// SIMATIC S7-200 project (STEP 7-Micro/WIN), CPU 224 REL 01.22

ORGANIZATION_BLOCK MAIN:OB1
TITLE=POU Comment
BEGIN
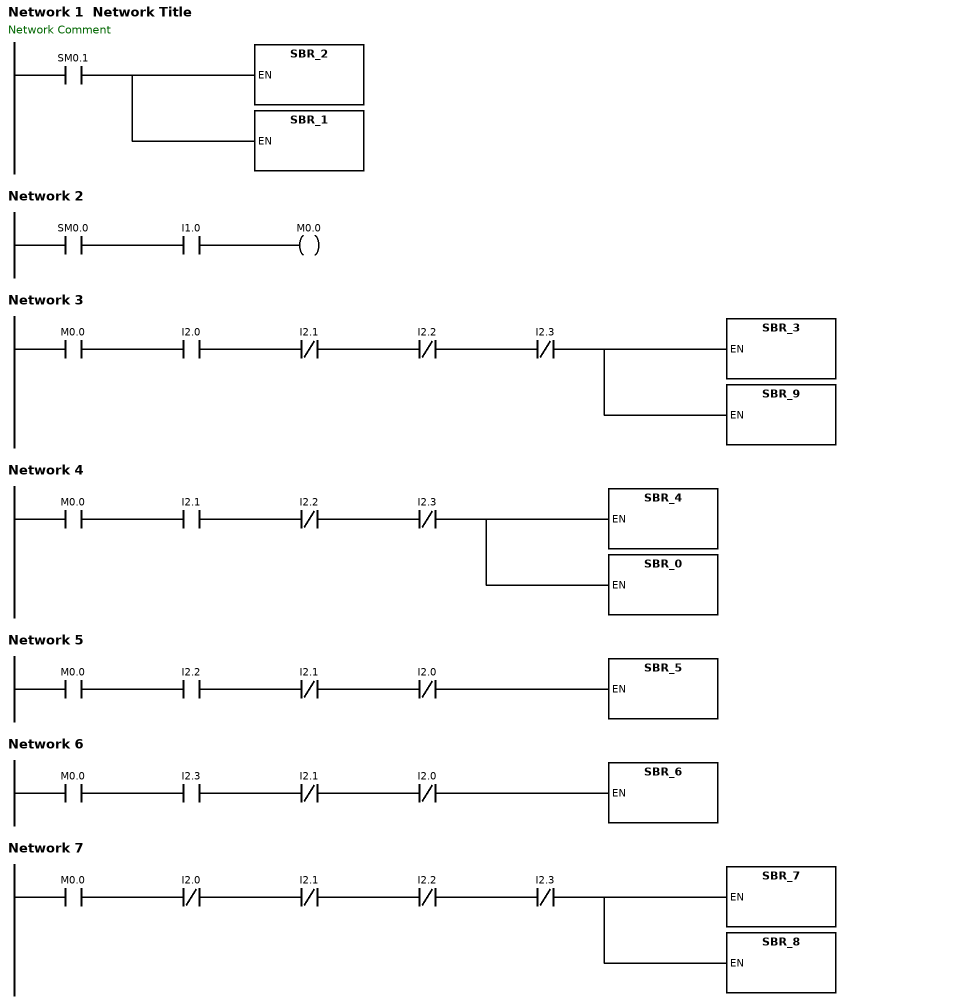
Network 1 // Network Title
// Network Comment
LD     SM0.1
CALL   SBR_2:SBR2
CALL   SBR_1:SBR1
Network 2
LD     SM0.0
A      I1.0
=      M0.0
Network 3
LD     M0.0
A      I2.0
AN     I2.1
AN     I2.2
AN     I2.3
CALL   SBR_3:SBR3
CALL   SBR_9:SBR9
Network 4
LD     M0.0
A      I2.1
AN     I2.2
AN     I2.3
CALL   SBR_4:SBR4
CALL   SBR_0:SBR0
Network 5
LD     M0.0
A      I2.2
AN     I2.1
AN     I2.0
CALL   SBR_5:SBR5
Network 6
LD     M0.0
A      I2.3
AN     I2.1
AN     I2.0
CALL   SBR_6:SBR6
Network 7
LD     M0.0
AN     I2.0
AN     I2.1
AN     I2.2
AN     I2.3
CALL   SBR_7:SBR7
CALL   SBR_8:SBR8
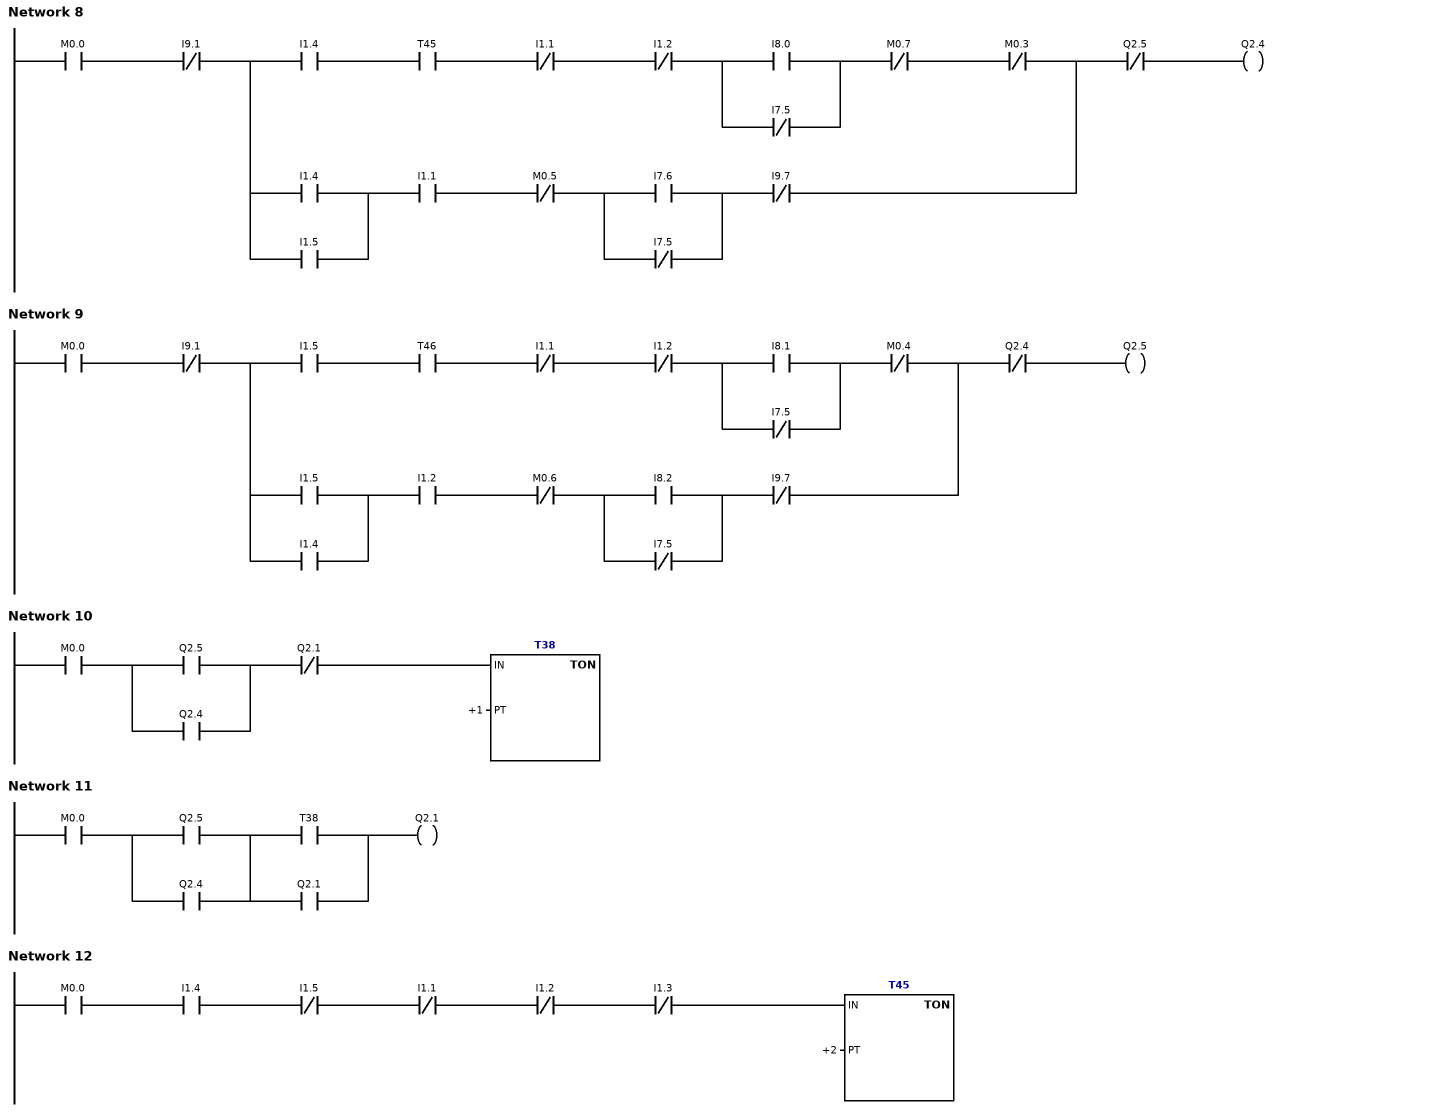
Network 8
LD     M0.0
AN     I9.1
LD     I1.4
A      T45
AN     I1.1
AN     I1.2
LD     I8.0
ON     I7.5
ALD
AN     M0.7
AN     M0.3
LD     I1.4
O      I1.5
A      I1.1
AN     M0.5
LD     I7.6
ON     I7.5
ALD
AN     I9.7
OLD
ALD
AN     Q2.5
=      Q2.4
Network 9
LD     M0.0
AN     I9.1
LD     I1.5
A      T46
AN     I1.1
AN     I1.2
LD     I8.1
ON     I7.5
ALD
AN     M0.4
LD     I1.5
O      I1.4
A      I1.2
AN     M0.6
LD     I8.2
ON     I7.5
ALD
AN     I9.7
OLD
ALD
AN     Q2.4
=      Q2.5
Network 10
LD     M0.0
LD     Q2.5
O      Q2.4
ALD
AN     Q2.1
TON    T38, +1
Network 11
LD     M0.0
LD     Q2.5
O      Q2.4
ALD
LD     T38
O      Q2.1
ALD
=      Q2.1
Network 12
LD     M0.0
A      I1.4
AN     I1.5
AN     I1.1
AN     I1.2
AN     I1.3
TON    T45, +2
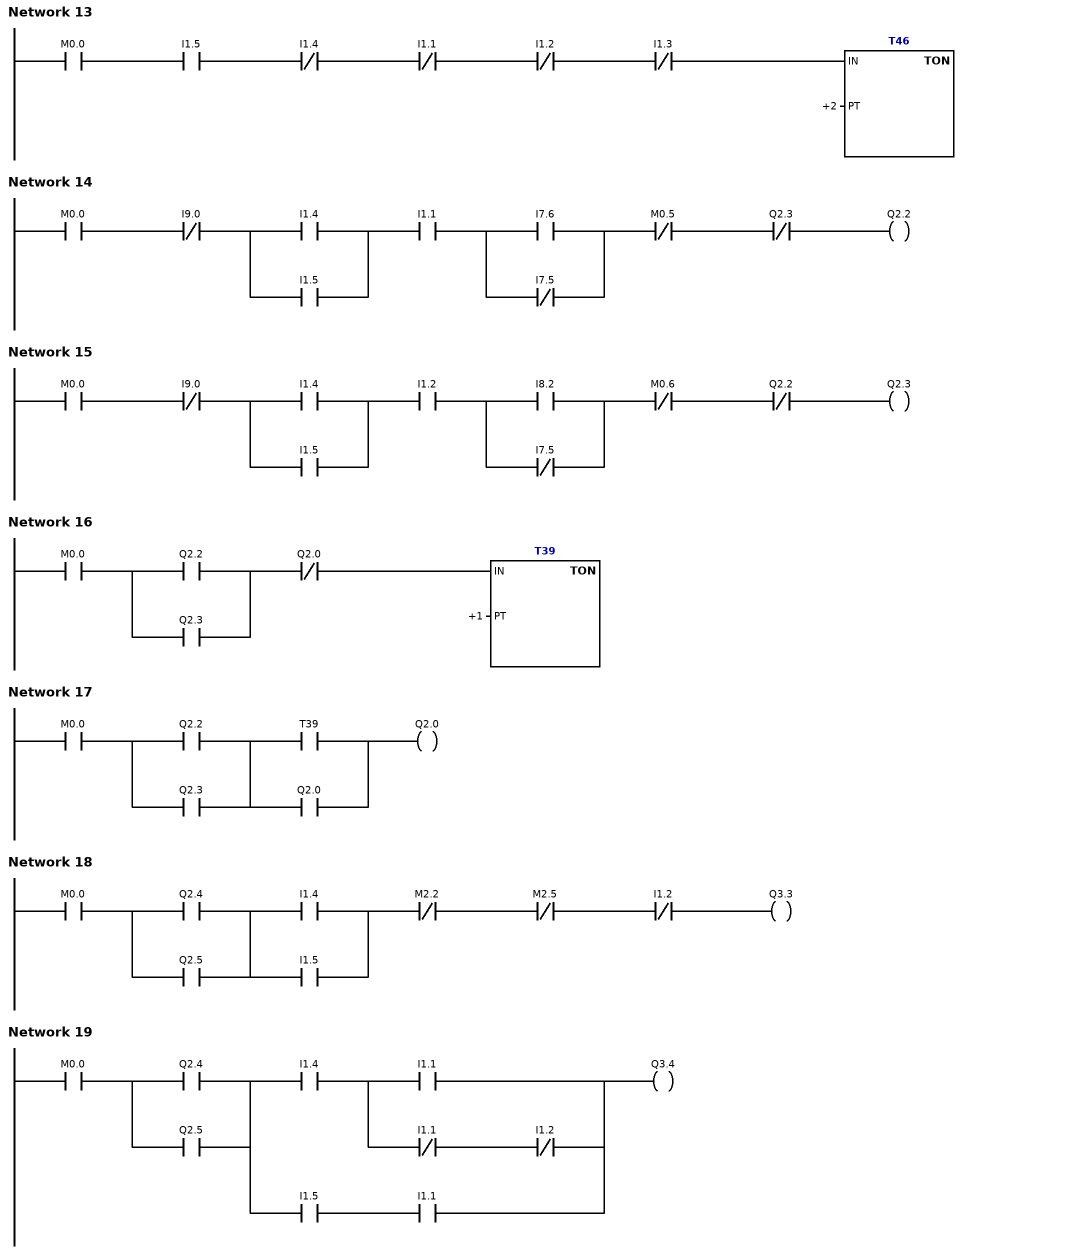
Network 13
LD     M0.0
A      I1.5
AN     I1.4
AN     I1.1
AN     I1.2
AN     I1.3
TON    T46, +2
Network 14
LD     M0.0
AN     I9.0
LD     I1.4
O      I1.5
ALD
A      I1.1
LD     I7.6
ON     I7.5
ALD
AN     M0.5
AN     Q2.3
=      Q2.2
Network 15
LD     M0.0
AN     I9.0
LD     I1.4
O      I1.5
ALD
A      I1.2
LD     I8.2
ON     I7.5
ALD
AN     M0.6
AN     Q2.2
=      Q2.3
Network 16
LD     M0.0
LD     Q2.2
O      Q2.3
ALD
AN     Q2.0
TON    T39, +1
Network 17
LD     M0.0
LD     Q2.2
O      Q2.3
ALD
LD     T39
O      Q2.0
ALD
=      Q2.0
Network 18
LD     M0.0
LD     Q2.4
O      Q2.5
ALD
LD     I1.4
O      I1.5
ALD
AN     M2.2
AN     M2.5
AN     I1.2
=      Q3.3
Network 19
LD     M0.0
LD     Q2.4
O      Q2.5
ALD
LD     I1.4
LD     I1.1
LDN    I1.1
AN     I1.2
OLD
ALD
LD     I1.5
A      I1.1
OLD
ALD
=      Q3.4
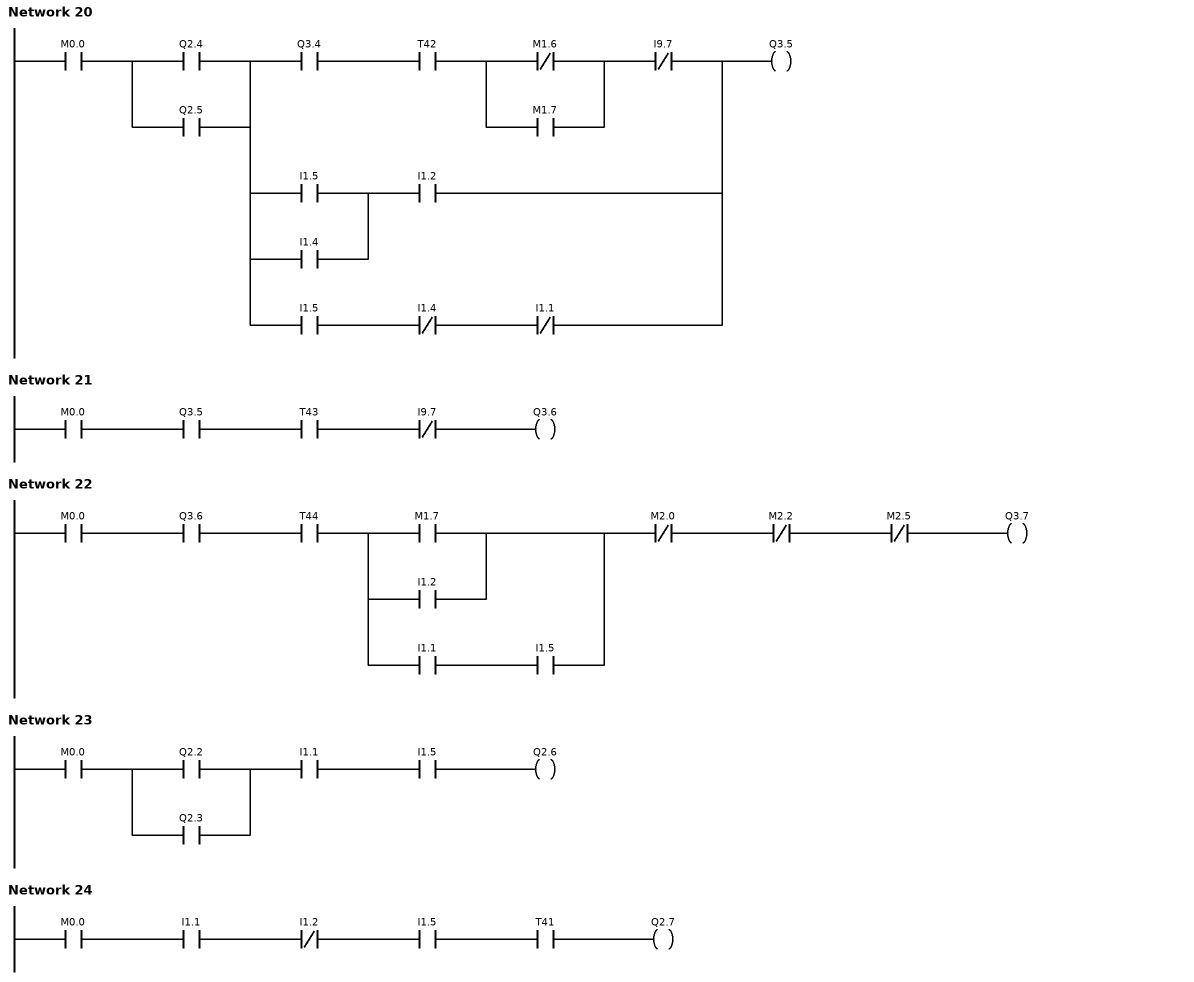
Network 20
LD     M0.0
LD     Q2.4
O      Q2.5
ALD
LD     Q3.4
A      T42
LDN    M1.6
O      M1.7
ALD
AN     I9.7
LD     I1.5
O      I1.4
A      I1.2
OLD
LD     I1.5
AN     I1.4
AN     I1.1
OLD
ALD
=      Q3.5
Network 21
LD     M0.0
A      Q3.5
A      T43
AN     I9.7
=      Q3.6
Network 22
LD     M0.0
A      Q3.6
A      T44
LD     M1.7
O      I1.2
LD     I1.1
A      I1.5
OLD
ALD
AN     M2.0
AN     M2.2
AN     M2.5
=      Q3.7
Network 23
LD     M0.0
LD     Q2.2
O      Q2.3
ALD
A      I1.1
A      I1.5
=      Q2.6
Network 24
LD     M0.0
A      I1.1
AN     I1.2
A      I1.5
A      T41
=      Q2.7
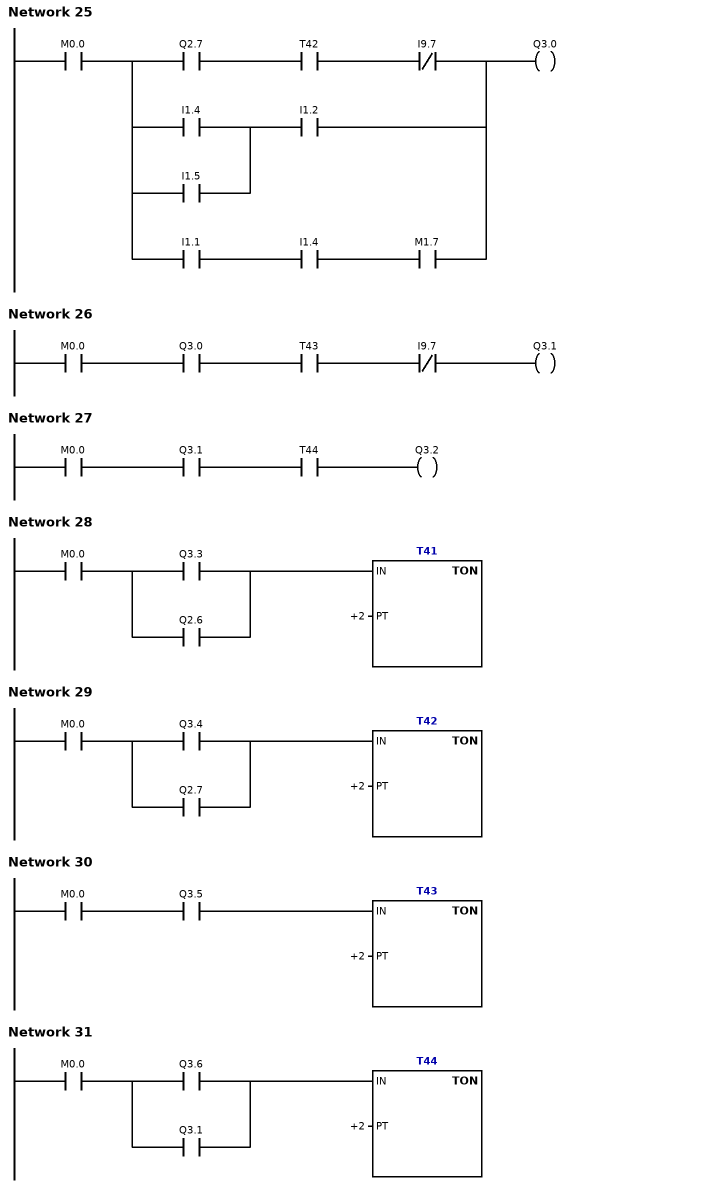
Network 25
LD     M0.0
LD     Q2.7
A      T42
AN     I9.7
LD     I1.4
O      I1.5
A      I1.2
OLD
LD     I1.1
A      I1.4
A      M1.7
OLD
ALD
=      Q3.0
Network 26
LD     M0.0
A      Q3.0
A      T43
AN     I9.7
=      Q3.1
Network 27
LD     M0.0
A      Q3.1
A      T44
=      Q3.2
Network 28
LD     M0.0
LD     Q3.3
O      Q2.6
ALD
TON    T41, +2
Network 29
LD     M0.0
LD     Q3.4
O      Q2.7
ALD
TON    T42, +2
Network 30
LD     M0.0
A      Q3.5
TON    T43, +2
Network 31
LD     M0.0
LD     Q3.6
O      Q3.1
ALD
TON    T44, +2
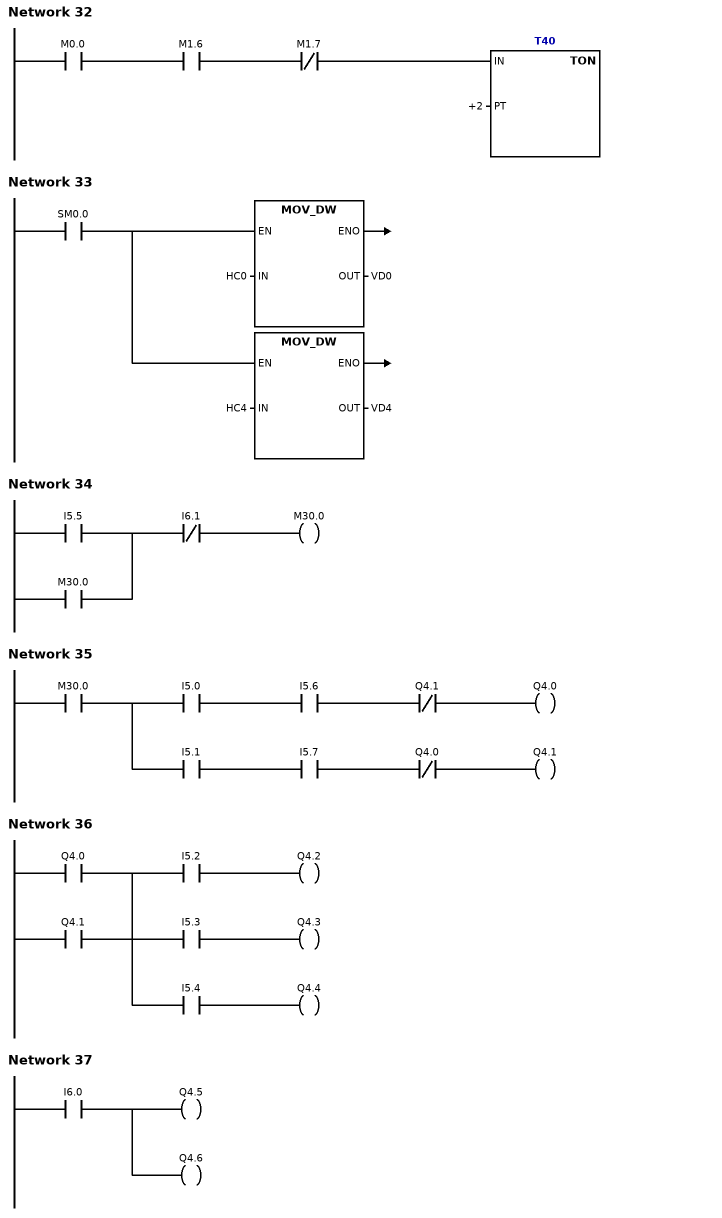
Network 32
LD     M0.0
A      M1.6
AN     M1.7
TON    T40, +2
Network 33
LD     SM0.0
MOVD   HC0, VD0
MOVD   HC4, VD4
Network 34
LD     I5.5
O      M30.0
AN     I6.1
=      M30.0
Network 35
LD     M30.0
LPS
A      I5.0
A      I5.6
AN     Q4.1
=      Q4.0
LPP
A      I5.1
A      I5.7
AN     Q4.0
=      Q4.1
Network 36
LD     Q4.0
O      Q4.1
LPS
A      I5.2
=      Q4.2
LRD
A      I5.3
=      Q4.3
LPP
A      I5.4
=      Q4.4
Network 37
LD     I6.0
=      Q4.5
=      Q4.6
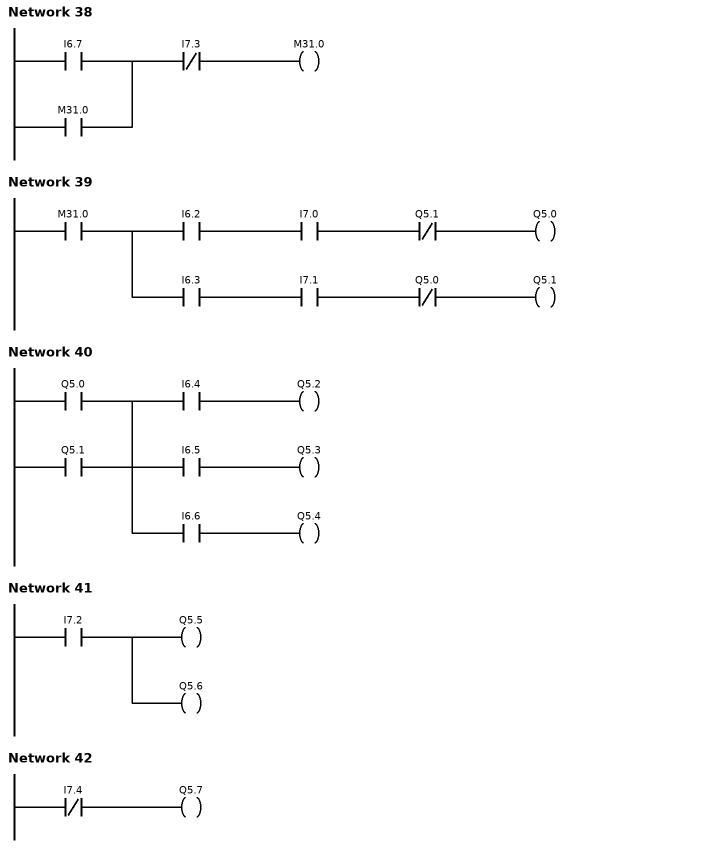
Network 38
LD     I6.7
O      M31.0
AN     I7.3
=      M31.0
Network 39
LD     M31.0
LPS
A      I6.2
A      I7.0
AN     Q5.1
=      Q5.0
LPP
A      I6.3
A      I7.1
AN     Q5.0
=      Q5.1
Network 40
LD     Q5.0
O      Q5.1
LPS
A      I6.4
=      Q5.2
LRD
A      I6.5
=      Q5.3
LPP
A      I6.6
=      Q5.4
Network 41
LD     I7.2
=      Q5.5
=      Q5.6
Network 42
LDN    I7.4
=      Q5.7
END_ORGANIZATION_BLOCK

SUBROUTINE_BLOCK SBR_0:SBR0
TITLE=POU Comment
BEGIN
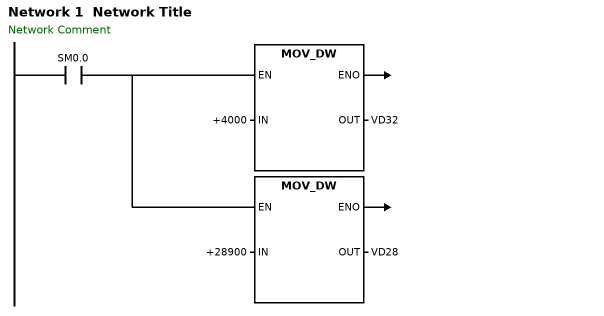
Network 1 // Network Title
// Network Comment
// (network saved uncompiled; LAD cells follow)
// row 0: c0 -| |- SM0.0 v  c1 --  c2 [MOV_DW EN:=power@row0, IN:=+4000, ENO=>power, OUT=>VD32]  c3 ->
// row 1: c0 ^v  c2 [box]
// row 2: c0 ^  c1 --  c2 [MOV_DW EN:=power@row2, IN:=+28900, ENO=>power, OUT=>VD28]  c3 ->
// row 3: c2 [box]
END_SUBROUTINE_BLOCK

SUBROUTINE_BLOCK SBR_1:SBR1
TITLE=
BEGIN
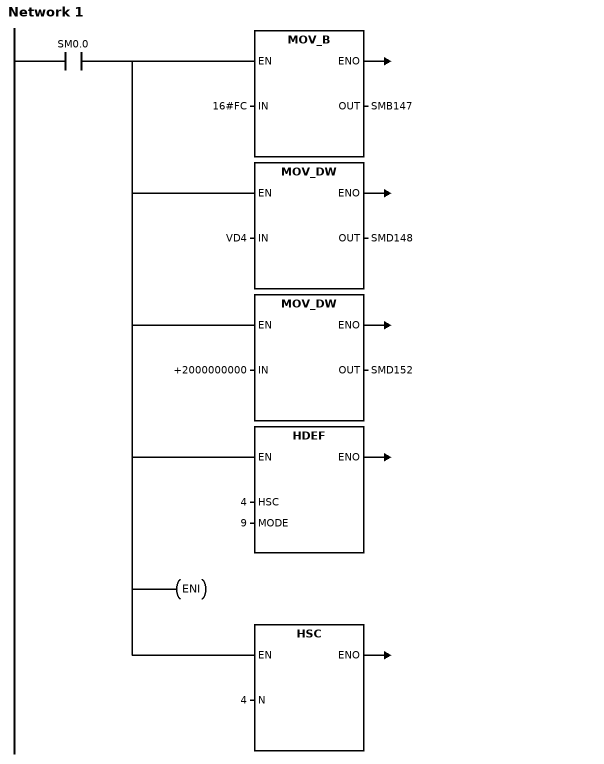
Network 1
// (network saved uncompiled; LAD cells follow)
// row 0: c0 -| |- SM0.0 v  c1 --  c2 [MOV_B EN:=power@row0, IN:=16#FC, ENO=>power, OUT=>SMB147]  c3 ->
// row 1: c0 ^v  c2 [box]
// row 2: c0 ^v  c1 --  c2 [MOV_DW EN:=power@row2, IN:=VD4, ENO=>power, OUT=>SMD148]  c3 ->
// row 3: c0 ^v  c2 [box]
// row 4: c0 ^v  c1 --  c2 [MOV_DW EN:=power@row4, IN:=+2000000000, ENO=>power, OUT=>SMD152]  c3 ->
// row 5: c0 ^v  c2 [box]
// row 6: c0 ^v  c1 --  c2 [HDEF EN:=power@row6, HSC:=4, MODE:=9, ENO=>power]  c3 ->
// row 7: c0 ^v  c2 [box]
// row 8: c0 ^v  c1 -(ENI)
// row 9: c0 ^  c1 --  c2 [HSC EN:=power@row9, N:=4, ENO=>power]  c3 ->
// row 10: c2 [box]
END_SUBROUTINE_BLOCK

SUBROUTINE_BLOCK SBR_2:SBR2
TITLE=
BEGIN
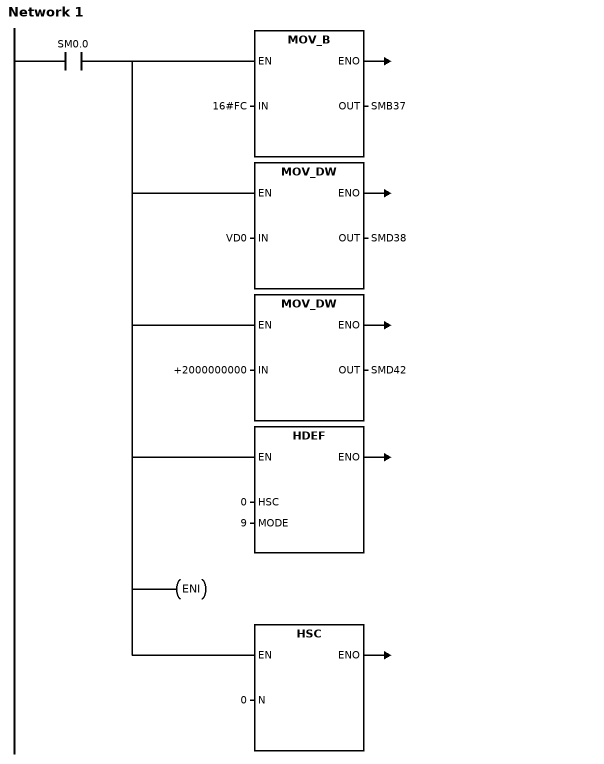
Network 1
// (network saved uncompiled; LAD cells follow)
// row 0: c0 -| |- SM0.0 v  c1 --  c2 [MOV_B EN:=power@row0, IN:=16#FC, ENO=>power, OUT=>SMB37]  c3 ->
// row 1: c0 ^v  c2 [box]
// row 2: c0 ^v  c1 --  c2 [MOV_DW EN:=power@row2, IN:=VD0, ENO=>power, OUT=>SMD38]  c3 ->
// row 3: c0 ^v  c2 [box]
// row 4: c0 ^v  c1 --  c2 [MOV_DW EN:=power@row4, IN:=+2000000000, ENO=>power, OUT=>SMD42]  c3 ->
// row 5: c0 ^v  c2 [box]
// row 6: c0 ^v  c1 --  c2 [HDEF EN:=power@row6, HSC:=0, MODE:=9, ENO=>power]  c3 ->
// row 7: c0 ^v  c2 [box]
// row 8: c0 ^v  c1 -(ENI)
// row 9: c0 ^  c1 --  c2 [HSC EN:=power@row9, N:=0, ENO=>power]  c3 ->
// row 10: c2 [box]
END_SUBROUTINE_BLOCK

SUBROUTINE_BLOCK SBR_3:SBR3
TITLE=
BEGIN
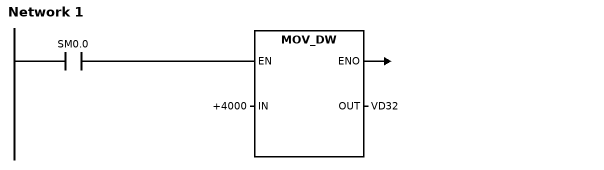
Network 1
// (network saved uncompiled; LAD cells follow)
// row 0: c0 -| |- SM0.0  c1 --  c2 [MOV_DW EN:=power@row0, IN:=+4000, ENO=>power, OUT=>VD32]  c3 ->
// row 1: c2 [box]
END_SUBROUTINE_BLOCK

SUBROUTINE_BLOCK SBR_4:SBR4
TITLE=
BEGIN
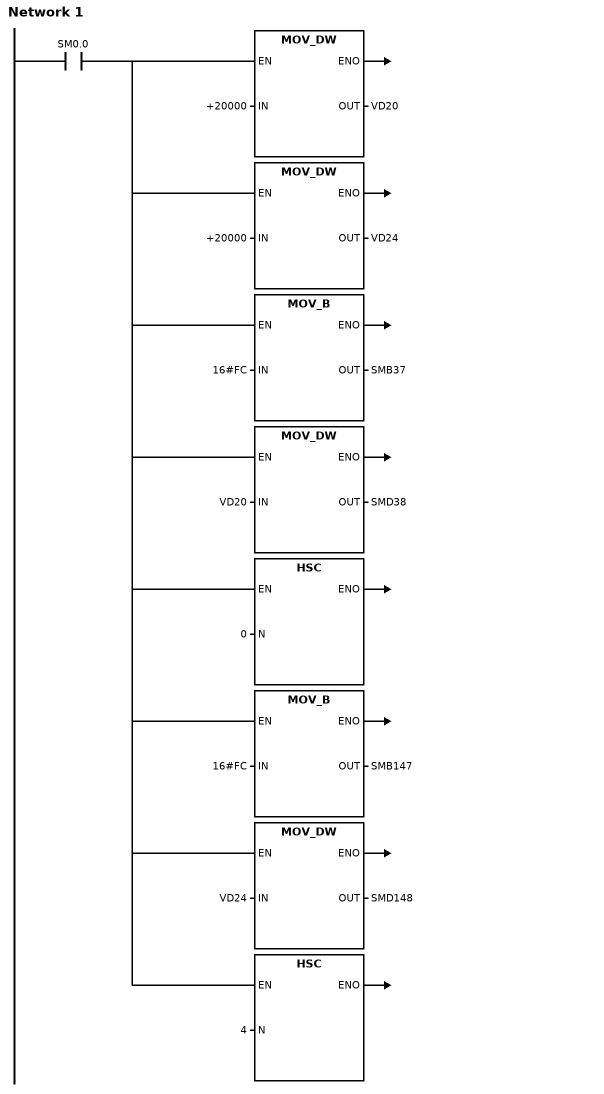
Network 1
// (network saved uncompiled; LAD cells follow)
// row 0: c0 -| |- SM0.0 v  c1 --  c2 [MOV_DW EN:=power@row0, IN:=+20000, ENO=>power, OUT=>VD20]  c3 ->
// row 1: c0 ^v  c2 [box]
// row 2: c0 ^v  c1 --  c2 [MOV_DW EN:=power@row2, IN:=+20000, ENO=>power, OUT=>VD24]  c3 ->
// row 3: c0 ^v  c2 [box]
// row 4: c0 ^v  c1 --  c2 [MOV_B EN:=power@row4, IN:=16#FC, ENO=>power, OUT=>SMB37]  c3 ->
// row 5: c0 ^v  c2 [box]
// row 6: c0 ^v  c1 --  c2 [MOV_DW EN:=power@row6, IN:=VD20, ENO=>power, OUT=>SMD38]  c3 ->
// row 7: c0 ^v  c2 [box]
// row 8: c0 ^v  c1 --  c2 [HSC EN:=power@row8, N:=0, ENO=>power]  c3 ->
// row 9: c0 ^v  c2 [box]
// row 10: c0 ^v  c1 --  c2 [MOV_B EN:=power@row10, IN:=16#FC, ENO=>power, OUT=>SMB147]  c3 ->
// row 11: c0 ^v  c2 [box]
// row 12: c0 ^v  c1 --  c2 [MOV_DW EN:=power@row12, IN:=VD24, ENO=>power, OUT=>SMD148]  c3 ->
// row 13: c0 ^v  c2 [box]
// row 14: c0 ^  c1 --  c2 [HSC EN:=power@row14, N:=4, ENO=>power]  c3 ->
// row 15: c2 [box]
END_SUBROUTINE_BLOCK

SUBROUTINE_BLOCK SBR_5:SBR5
TITLE=
BEGIN
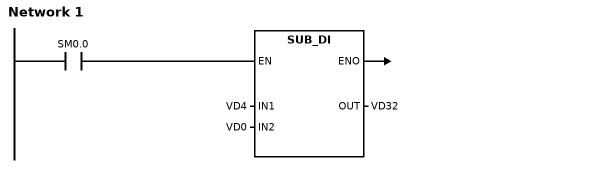
Network 1
// (network saved uncompiled; LAD cells follow)
// row 0: c0 -| |- SM0.0  c1 --  c2 [SUB_DI EN:=power@row0, IN1:=VD4, IN2:=VD0, ENO=>power, OUT=>VD32]  c3 ->
// row 1: c2 [box]
END_SUBROUTINE_BLOCK

SUBROUTINE_BLOCK SBR_6:SBR6
TITLE=
BEGIN
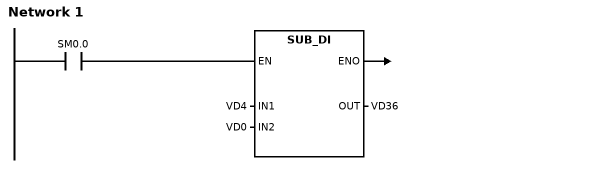
Network 1
// (network saved uncompiled; LAD cells follow)
// row 0: c0 -| |- SM0.0  c1 --  c2 [SUB_DI EN:=power@row0, IN1:=VD4, IN2:=VD0, ENO=>power, OUT=>VD36]  c3 ->
// row 1: c2 [box]
END_SUBROUTINE_BLOCK

SUBROUTINE_BLOCK SBR_7:SBR7
TITLE=
BEGIN
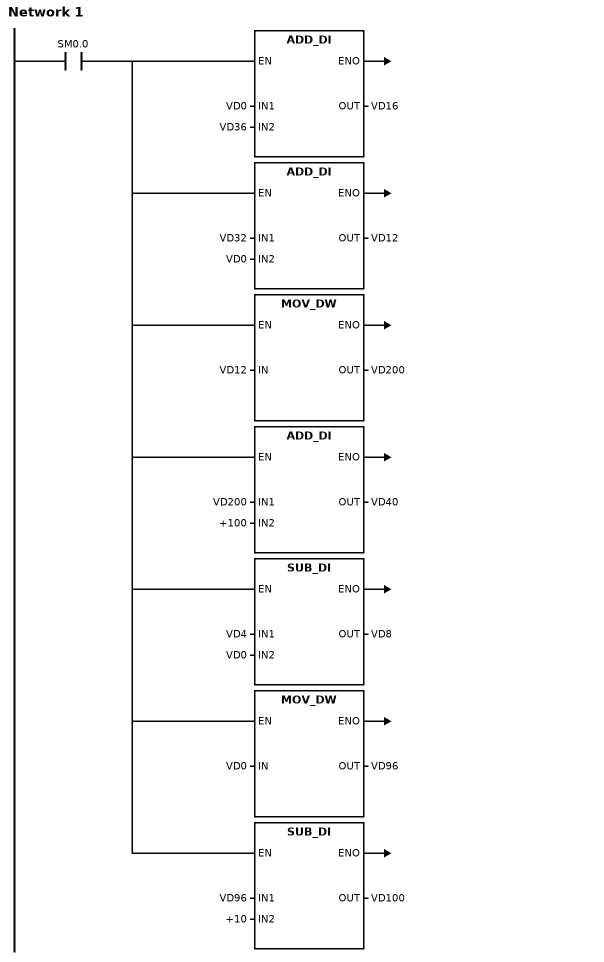
Network 1
// (network saved uncompiled; LAD cells follow)
// row 0: c0 -| |- SM0.0 v  c1 --  c2 [ADD_DI EN:=power@row0, IN1:=VD0, IN2:=VD36, ENO=>power, OUT=>VD16]  c3 ->
// row 1: c0 ^v  c2 [box]
// row 2: c0 ^v  c1 --  c2 [ADD_DI EN:=power@row2, IN1:=VD32, IN2:=VD0, ENO=>power, OUT=>VD12]  c3 ->
// row 3: c0 ^v  c2 [box]
// row 4: c0 ^v  c1 --  c2 [MOV_DW EN:=power@row4, IN:=VD12, ENO=>power, OUT=>VD200]  c3 ->
// row 5: c0 ^v  c2 [box]
// row 6: c0 ^v  c1 --  c2 [ADD_DI EN:=power@row6, IN1:=VD200, IN2:=+100, ENO=>power, OUT=>VD40]  c3 ->
// row 7: c0 ^v  c2 [box]
// row 8: c0 ^v  c1 --  c2 [SUB_DI EN:=power@row8, IN1:=VD4, IN2:=VD0, ENO=>power, OUT=>VD8]  c3 ->
// row 9: c0 ^v  c2 [box]
// row 10: c0 ^v  c1 --  c2 [MOV_DW EN:=power@row10, IN:=VD0, ENO=>power, OUT=>VD96]  c3 ->
// row 11: c0 ^v  c2 [box]
// row 12: c0 ^  c1 --  c2 [SUB_DI EN:=power@row12, IN1:=VD96, IN2:=+10, ENO=>power, OUT=>VD100]  c3 ->
// row 13: c2 [box]
END_SUBROUTINE_BLOCK

SUBROUTINE_BLOCK SBR_8:SBR8
TITLE=POU Comment
BEGIN
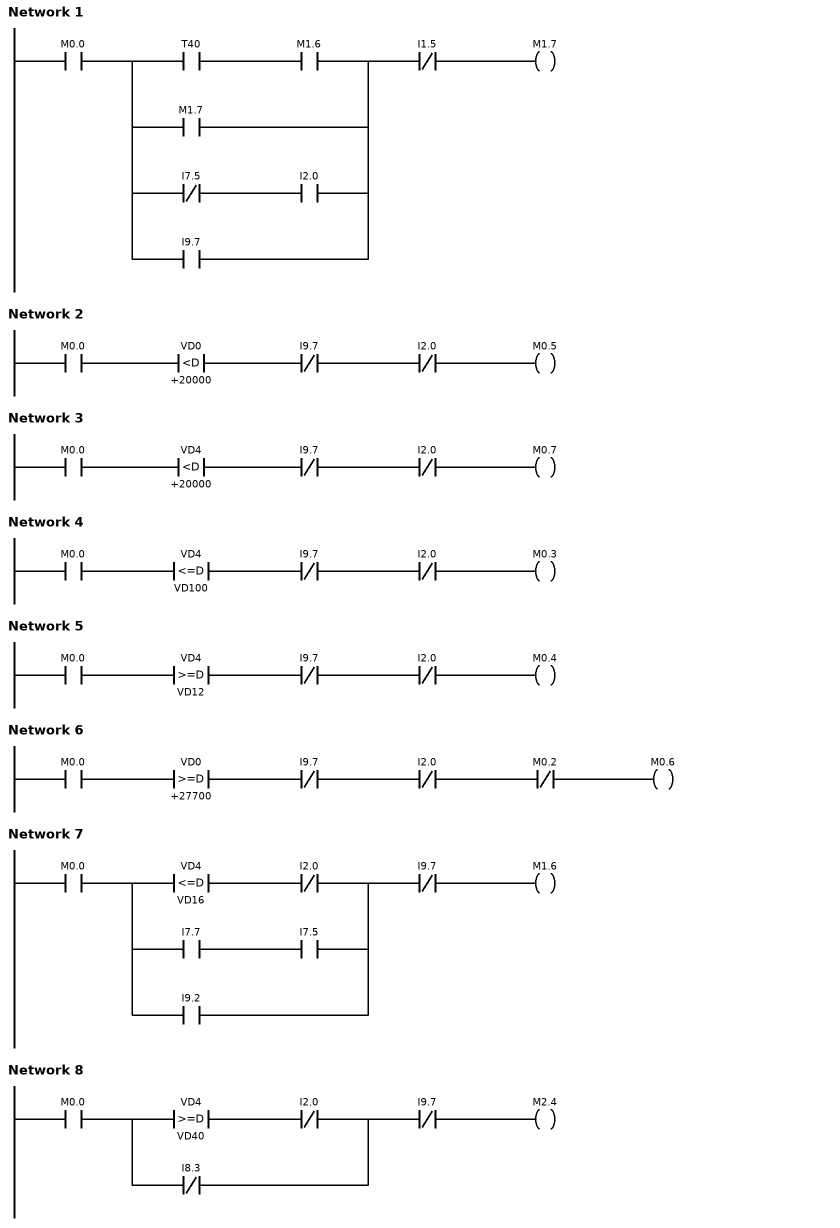
Network 1
// (network saved uncompiled; LAD cells follow)
// row 0: c0 -| |- M0.0 v  c1 -| |- T40  c2 -| |- M1.6 v  c3 -|/|- I1.5  c4 -( ) M1.7
// row 1: c0 ^v  c1 -| |- M1.7  c2 -- ^v
// row 2: c0 ^v  c1 -|/|- I7.5  c2 -| |- I2.0 ^v
// row 3: c0 ^  c1 -| |- I9.7  c2 -- ^
Network 2
// (network saved uncompiled; LAD cells follow)
// row 0: c0 -| |- M0.0  c1 -|<D|- VD0, +20000  c2 -|/|- I9.7  c3 -|/|- I2.0  c4 -( ) M0.5
Network 3
// (network saved uncompiled; LAD cells follow)
// row 0: c0 -| |- M0.0  c1 -|<D|- VD4, +20000  c2 -|/|- I9.7  c3 -|/|- I2.0  c4 -( ) M0.7
Network 4
// (network saved uncompiled; LAD cells follow)
// row 0: c0 -| |- M0.0  c1 -|<=D|- VD4, VD100  c2 -|/|- I9.7  c3 -|/|- I2.0  c4 -( ) M0.3
Network 5
// (network saved uncompiled; LAD cells follow)
// row 0: c0 -| |- M0.0  c1 -|>=D|- VD4, VD12  c2 -|/|- I9.7  c3 -|/|- I2.0  c4 -( ) M0.4
Network 6
// (network saved uncompiled; LAD cells follow)
// row 0: c0 -| |- M0.0  c1 -|>=D|- VD0, +27700  c2 -|/|- I9.7  c3 -|/|- I2.0  c4 -|/|- M0.2  c5 -( ) M0.6
Network 7
// (network saved uncompiled; LAD cells follow)
// row 0: c0 -| |- M0.0 v  c1 -|<=D|- VD4, VD16  c2 -|/|- I2.0 v  c3 -|/|- I9.7  c4 -( ) M1.6
// row 1: c0 ^v  c1 -| |- I7.7  c2 -| |- I7.5 ^v
// row 2: c0 ^  c1 -| |- I9.2  c2 -- ^
Network 8
// (network saved uncompiled; LAD cells follow)
// row 0: c0 -| |- M0.0 v  c1 -|>=D|- VD4, VD40  c2 -|/|- I2.0 v  c3 -|/|- I9.7  c4 -( ) M2.4
// row 1: c0 ^  c1 -|/|- I8.3  c2 -- ^
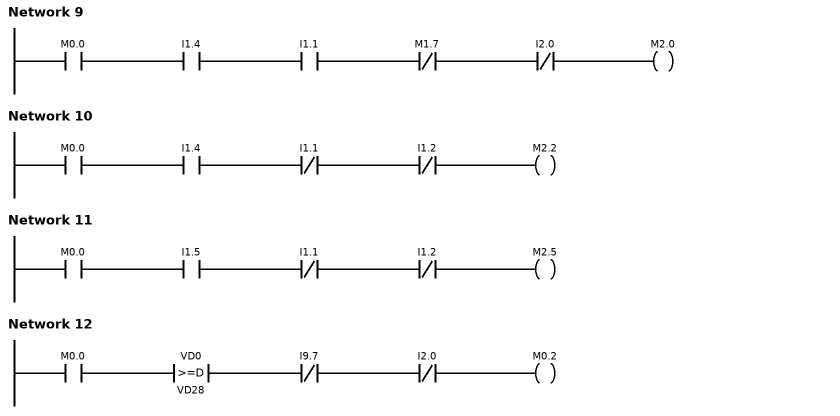
Network 9
// (network saved uncompiled; LAD cells follow)
// row 0: c0 -| |- M0.0  c1 -| |- I1.4  c2 -| |- I1.1  c3 -|/|- M1.7  c4 -|/|- I2.0  c5 -( ) M2.0
Network 10
// (network saved uncompiled; LAD cells follow)
// row 0: c0 -| |- M0.0  c1 -| |- I1.4  c2 -|/|- I1.1  c3 -|/|- I1.2  c4 -( ) M2.2
Network 11
// (network saved uncompiled; LAD cells follow)
// row 0: c0 -| |- M0.0  c1 -| |- I1.5  c2 -|/|- I1.1  c3 -|/|- I1.2  c4 -( ) M2.5
Network 12
// (network saved uncompiled; LAD cells follow)
// row 0: c0 -| |- M0.0  c1 -|>=D|- VD0, VD28  c2 -|/|- I9.7  c3 -|/|- I2.0  c4 -( ) M0.2
Network 13 // Network Title
// Network Comment
END_SUBROUTINE_BLOCK

SUBROUTINE_BLOCK SBR_9:SBR9
TITLE=POU Comment
BEGIN
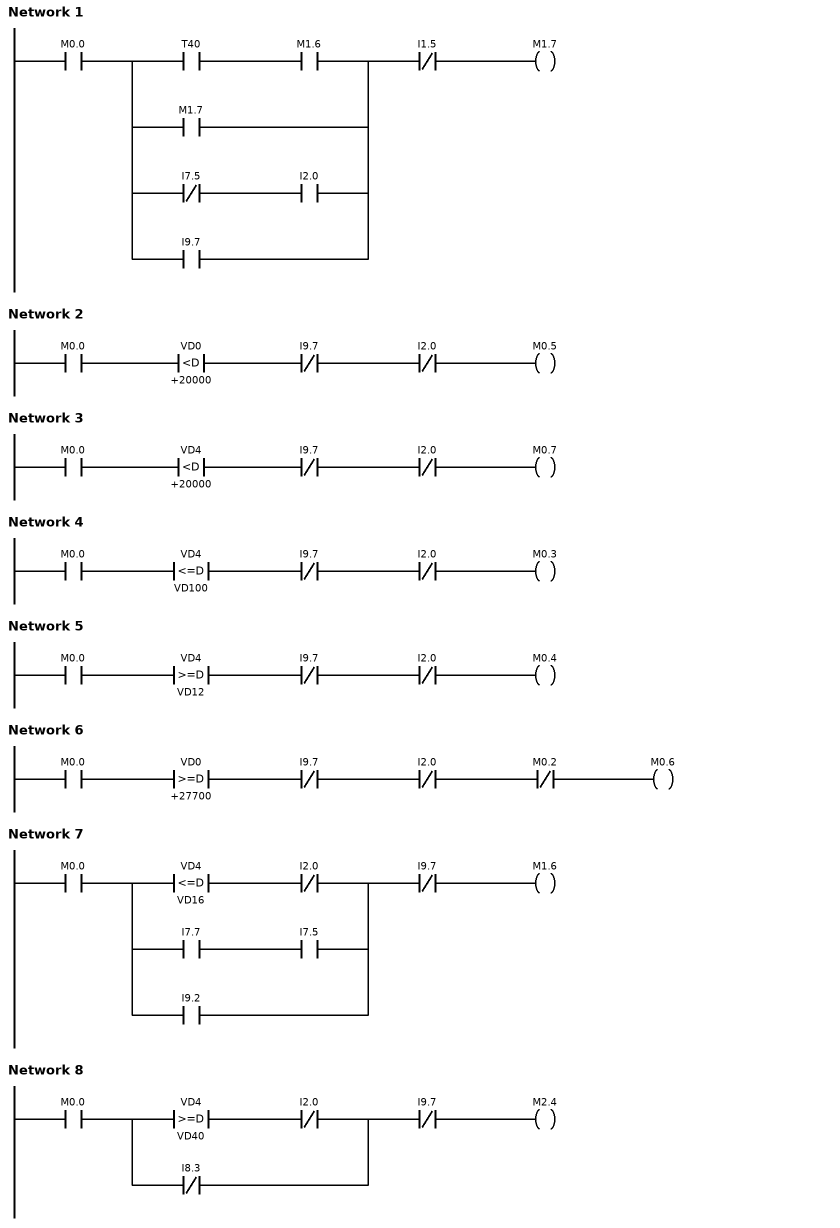
Network 1
// (network saved uncompiled; LAD cells follow)
// row 0: c0 -| |- M0.0 v  c1 -| |- T40  c2 -| |- M1.6 v  c3 -|/|- I1.5  c4 -( ) M1.7
// row 1: c0 ^v  c1 -| |- M1.7  c2 -- ^v
// row 2: c0 ^v  c1 -|/|- I7.5  c2 -| |- I2.0 ^v
// row 3: c0 ^  c1 -| |- I9.7  c2 -- ^
Network 2
// (network saved uncompiled; LAD cells follow)
// row 0: c0 -| |- M0.0  c1 -|<D|- VD0, +20000  c2 -|/|- I9.7  c3 -|/|- I2.0  c4 -( ) M0.5
Network 3
// (network saved uncompiled; LAD cells follow)
// row 0: c0 -| |- M0.0  c1 -|<D|- VD4, +20000  c2 -|/|- I9.7  c3 -|/|- I2.0  c4 -( ) M0.7
Network 4
// (network saved uncompiled; LAD cells follow)
// row 0: c0 -| |- M0.0  c1 -|<=D|- VD4, VD100  c2 -|/|- I9.7  c3 -|/|- I2.0  c4 -( ) M0.3
Network 5
// (network saved uncompiled; LAD cells follow)
// row 0: c0 -| |- M0.0  c1 -|>=D|- VD4, VD12  c2 -|/|- I9.7  c3 -|/|- I2.0  c4 -( ) M0.4
Network 6
// (network saved uncompiled; LAD cells follow)
// row 0: c0 -| |- M0.0  c1 -|>=D|- VD0, +27700  c2 -|/|- I9.7  c3 -|/|- I2.0  c4 -|/|- M0.2  c5 -( ) M0.6
Network 7
// (network saved uncompiled; LAD cells follow)
// row 0: c0 -| |- M0.0 v  c1 -|<=D|- VD4, VD16  c2 -|/|- I2.0 v  c3 -|/|- I9.7  c4 -( ) M1.6
// row 1: c0 ^v  c1 -| |- I7.7  c2 -| |- I7.5 ^v
// row 2: c0 ^  c1 -| |- I9.2  c2 -- ^
Network 8
// (network saved uncompiled; LAD cells follow)
// row 0: c0 -| |- M0.0 v  c1 -|>=D|- VD4, VD40  c2 -|/|- I2.0 v  c3 -|/|- I9.7  c4 -( ) M2.4
// row 1: c0 ^  c1 -|/|- I8.3  c2 -- ^
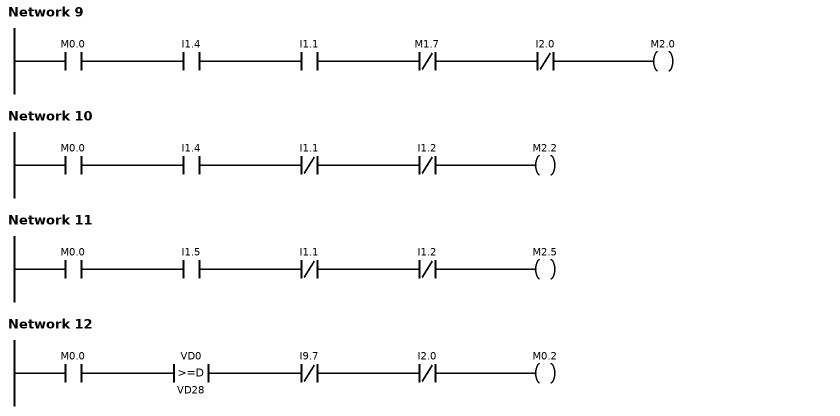
Network 9
// (network saved uncompiled; LAD cells follow)
// row 0: c0 -| |- M0.0  c1 -| |- I1.4  c2 -| |- I1.1  c3 -|/|- M1.7  c4 -|/|- I2.0  c5 -( ) M2.0
Network 10
// (network saved uncompiled; LAD cells follow)
// row 0: c0 -| |- M0.0  c1 -| |- I1.4  c2 -|/|- I1.1  c3 -|/|- I1.2  c4 -( ) M2.2
Network 11
// (network saved uncompiled; LAD cells follow)
// row 0: c0 -| |- M0.0  c1 -| |- I1.5  c2 -|/|- I1.1  c3 -|/|- I1.2  c4 -( ) M2.5
Network 12
// (network saved uncompiled; LAD cells follow)
// row 0: c0 -| |- M0.0  c1 -|>=D|- VD0, VD28  c2 -|/|- I9.7  c3 -|/|- I2.0  c4 -( ) M0.2
Network 13 // Network Title
// Network Comment
Network 21 // Network Title
// Network Comment
END_SUBROUTINE_BLOCK
